// TIA Portal V19 export
DATA_BLOCK "SUGAR TRANSFER CYCLE DB"   // DB100
{ S7_Optimized_Access := 'TRUE' }
// stored: MemoryReserve 100
   VAR RETAIN
      TRANSFER : Struct
         "TRANSFER START" : Bool;
         "TRANSFER STOP" : Bool;
         "TRANSFER OVER" : Bool;
         "TRANSFER BUFF" : Struct
            "SUGAR TO PREMIXING" : Int;
            "SUGAR TO MFG" : Int;
         END_STRUCT;
         SELECT : Struct
            "SUGAR TO PREMIXING" : Bool;
            "SUGAR TO MFG" : Bool;
            "SELECT BUFF" : Int;
         END_STRUCT;
      END_STRUCT;
      "SET PARAMETER" : Struct
         "SUGAR TO PREMIXING" : Real;
         "SUGAR TO MFG" : Real;
         "SET TIME" : Struct
            "SUGAR TO PREMIXING" : Int;
            "SUGAR TO MFG" : Int;
         END_STRUCT;
         RPM : Struct
            "SUGAR TO PREMIXING" : Real;
            "SUGAR TO MFG" : Real;
         END_STRUCT;
      END_STRUCT;
      "PV PARAMETER" : Struct
         "SUGAR TO PREMIXING" : Real;
         "SUGAR TO MFG" : Real;
         "PV TIME" : Struct
            "SUGAR TO PREMIXING" : Int;
            "SUGAR TO MFG" : Int;
         END_STRUCT;
      END_STRUCT;
   END_VAR
BEGIN
END_DATA_BLOCK
